FUNCTION_BLOCK FB_TelescopeTrackingState EXTENDS FB_TelescopeState
VAR_INPUT
END_VAR
VAR_OUTPUT
END_VAR
VAR
	pMachine : POINTER TO FB_TelescopeMachine;
END_VAR

METHOD FB_init : BOOL
VAR_INPUT
	bInitRetains : BOOL; // if TRUE, the retain variables are initialized (warm start / cold start)
	bInCopyCode : BOOL;  // if TRUE, the instance afterwards gets moved into the copy code (online change)
	pMachine : POINTER TO FB_TelescopeMachine;
END_VAR
THIS^.pMachine := pMachine;
END_METHOD

METHOD Park : BOOL
VAR_INPUT
END_VAR
END_METHOD

METHOD Slew : BOOL
VAR_INPUT
	fAzimuth	: LREAL;
	fAltitude	: LREAL;
END_VAR
END_METHOD

METHOD Stop : BOOL
VAR_INPUT
END_VAR
END_METHOD

METHOD Track : BOOL
VAR_INPUT
	fRightAscension	: LREAL;
	fDeclination	: LREAL;
END_VAR
END_METHOD

END_FUNCTION_BLOCK

(* stored: Version 1.1.0.1, ProductVersion 3.1.4024.15
   POU FB_TelescopeTrackingState: Id {436998b5-026e-41ee-9964-5eadbd61b386}, SpecialFunc None
   Method FB_init: Id {85c79bd5-8c18-466d-9f40-a59ddf3e019f}
   Method Park: Id {ab2d278a-f6a1-455c-971a-220210dec268}
   Method Slew: Id {711baa5c-acc3-43a5-947a-f41614b97294}
   Method Stop: Id {52d33a34-7731-4a63-a56d-e9297b9bc334}
   Method Track: Id {9cf2bc44-0f8a-4eca-b0b1-f2d3a353f164} *)
